{attribute addProperty BoxType "AX8620-1000-0026"}
{attribute addProperty Id "PSM_PSM_StatuswordAT %I*PSM_PSM_Statusword_32E7AA9A1620WcStateAT %I*WcState_F855686C1620InfoDataAT %I*InfoData_0BDED7BF144180"}
{attribute addProperty CRC "2634610164"}
{attribute addProperty SizeInBites "176"}
{attribute addProperty SizeInBytes "22"}
TYPE AX8620_79E0BBE6 :
STRUCT
	{attribute addProperty Name "PSM_PSM_Statusword"}
	PSM_PSM_Statusword : PSM_PSM_Statusword_32E7AA9A;
	{attribute addProperty Name "WcState"}
	WcState : WcState_F855686C;
	{attribute addProperty Name "InfoData"}
	InfoData : InfoData_0BDED7BF;
END_STRUCT
END_TYPE

(* stored: Version 1.2.0.0, ProductVersion 3.1.4024.9
   DUT AX8620_79E0BBE6: Id {45900da1-451d-45ee-8c39-aff55c8b8668} *)
